ABB RAPID module: Module1.mod

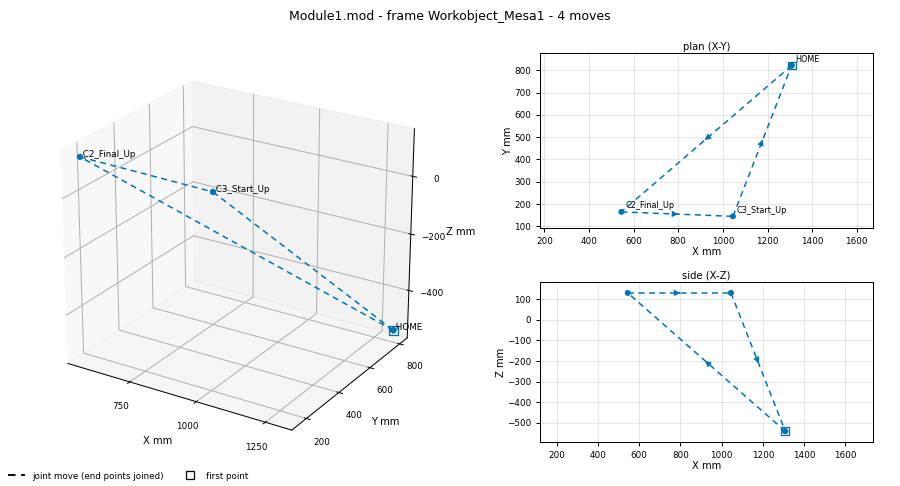
[picture p0: tool path of Module1.mod in frame Workobject_Mesa1, 4 of 4 moves have a stored position in this frame; points joined in program order, loops and branches not executed]
MODULE Module1
	CONST robtarget HOME:=[[1308.063364957,821.064844254,-540],[0.458291086,-0.458291086,0.538487958,-0.538487958],[0,0,0,0],[9E+09,9E+09,9E+09,9E+09,9E+09,9E+09]];
	CONST robtarget C1_Start_Up:=[[545,165,-130],[0.5,0.5,0.5,-0.5],[-2,-2,1,1],[9E+09,9E+09,9E+09,9E+09,9E+09,9E+09]];
	CONST robtarget C1_Start:=[[545,65,-130],[0.5,0.5,0.5,-0.5],[-2,-2,1,1],[9E+09,9E+09,9E+09,9E+09,9E+09,9E+09]];
	CONST robtarget C1_Final:=[[545,65,-100],[0.5,0.5,0.5,-0.5],[-2,-2,1,1],[9E+09,9E+09,9E+09,9E+09,9E+09,9E+09]];
	CONST robtarget C1_Final_Up:=[[545,165,-100],[0.5,0.5,0.5,-0.5],[-2,-2,1,1],[9E+09,9E+09,9E+09,9E+09,9E+09,9E+09]];
	CONST robtarget C2_Start_Up:=[[545,165,100],[0.5,0.5,0.5,-0.5],[-2,-2,1,1],[9E+09,9E+09,9E+09,9E+09,9E+09,9E+09]];
	CONST robtarget C2_Start:=[[545,65,100],[0.5,0.5,0.5,-0.5],[-2,-2,1,1],[9E+09,9E+09,9E+09,9E+09,9E+09,9E+09]];
	CONST robtarget C2_Final:=[[545,65,130],[0.5,0.5,0.5,-0.5],[-2,-2,1,1],[9E+09,9E+09,9E+09,9E+09,9E+09,9E+09]];
	CONST robtarget C2_Final_Up:=[[545,165,130],[0.5,0.5,0.5,-0.5],[-2,-2,1,1],[9E+09,9E+09,9E+09,9E+09,9E+09,9E+09]];
	CONST robtarget C3_Start_Up:=[[1045,145,130],[0.5,0.5,0.5,-0.5],[0,0,0,0],[9E+09,9E+09,9E+09,9E+09,9E+09,9E+09]];
	CONST robtarget C3_Start:=[[1045,65,130],[0.5,0.5,0.5,-0.5],[0,0,0,0],[9E+09,9E+09,9E+09,9E+09,9E+09,9E+09]];
	CONST robtarget C3_Final:=[[1045,65,100],[0.5,0.5,0.5,-0.5],[0,0,0,0],[9E+09,9E+09,9E+09,9E+09,9E+09,9E+09]];
	CONST robtarget C3_Final_Up:=[[1045,165,100],[0.5,0.5,0.5,-0.5],[0,0,0,0],[9E+09,9E+09,9E+09,9E+09,9E+09,9E+09]];
	CONST robtarget C4_Start_Up:=[[1045,165,-100],[0.5,0.5,0.5,-0.5],[0,0,0,0],[9E+09,9E+09,9E+09,9E+09,9E+09,9E+09]];
	CONST robtarget C4_Start:=[[1045,65,-100],[0.5,0.5,0.5,-0.5],[0,0,0,0],[9E+09,9E+09,9E+09,9E+09,9E+09,9E+09]];
	CONST robtarget C4_Final:=[[1045,65,-130],[0.5,0.5,0.5,-0.5],[0,0,0,0],[9E+09,9E+09,9E+09,9E+09,9E+09,9E+09]];
	CONST robtarget C4_Final_Up:=[[1045,165,-130],[0.5,0.5,0.5,-0.5],[0,0,0,0],[9E+09,9E+09,9E+09,9E+09,9E+09,9E+09]];
    !***********************************************************
    !
    ! Module:  Module1
    !
    ! Description:
    !   <Insert description here>
    !
    ! Author: juanc
    !
    ! Version: 1.0
    !
    !***********************************************************


    !***********************************************************
    !
    ! Procedure main
    !
    !   This is the entry point of your program
    !
    !***********************************************************
    PROC main()
        BOCARRIBA_1;
    ENDPROC
	PROC BOCARRIBA_1()
	    MoveJ HOME,v1000,z100,AW_Gun\WObj:=Workobject_Mesa1;
	    MoveJ C2_Final_Up,v1000,z100,AW_Gun\WObj:=Workobject_Mesa1;
	    MoveJ C3_Start_Up,v200,z100,AW_Gun\WObj:=Workobject_Mesa1;
	    MoveJ HOME,v1000,z100,AW_Gun\WObj:=Workobject_Mesa1;
	ENDPROC
ENDMODULE
